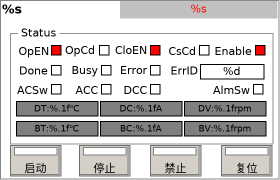
VISUALIZATION VPEModuleVis  // 280x180
VAR_IN_OUT
	userData: VPEHMIStruts;
END_VAR
    Button (10,145 51x31), "启动", input disabled if: NOT userData.HMIEnable
        tap userData.open
    Rectangle (14,147 43x8), colour toggle: userData.openRelay
    GroupBox (10,25 263x119), "Status"
        RoundedRectangle (41,40 10x10), colour toggle: userData.done
        RoundedRectangle (245,20 10x10), colour toggle: userData.enable
        RoundedRectangle (91,40 10x10), colour toggle: userData.busy
        RoundedRectangle (140,40 10x10), colour toggle: userData.error
        Rectangle (190,39 64x15), "%d", text variable: userData.errID
        Label (5,20 37x13), "OpEN"
        RoundedRectangle (41,20 10x10), colour toggle: userData.enableOpen
        RoundedRectangle (140,20 10x10), colour toggle: userData.enableClose
        Label (206,20 39x13), "Enable"
        Label (158,39 33x14), "ErrID"
        Label (110,39 30x13), "Error"
        Label (61,39 30x13), "Busy"
        Label (8,38 33x16), "Done"
        RoundedRectangle (41,59 10x10), colour toggle: userData.AccAprSw
        Label (203,59 40x13), "AlmSw"
        RoundedRectangle (243,59 10x10), colour toggle: userData.AlmAprSw
        Rectangle (6,96 82x15), "BT:%.1f℃", text variable: userData.BoosterTemperature, input disabled if: true
        RoundedRectangle (140,59 10x10), colour toggle: userData.Dccing
        RoundedRectangle (91,59 10x10), colour toggle: userData.Accing
        Label (52,19 36x13), "OpCd"
        RoundedRectangle (89,20 10x10), colour toggle: userData.opencondition
        Label (103,19 37x13), "CloEN"
    Button (221,145 51x31), "复位"
        tap userData.reset
    Rectangle (225,147 43x8), colour toggle: userData.reset
    Rectangle (-1,-1 119x20), "%s", text variable: userData.nameTXT
    Button (79,145 51x31), "停止"
        tap userData.close
    Rectangle (83,147 43x8)
    Label (14,84 37x13), "ACSw"
    Button (150,145 51x31), "禁止"
        tap userData.stop
    Rectangle (16,101 82x15), "DT:%.1f℃", text variable: userData.DryPumpTemperature, input disabled if: true
    Rectangle (100,101 82x15), "DC:%.1fA", text variable: userData.DryPumpCurrent, input disabled if: true
    Rectangle (184,101 82x15), "DV:%.1frpm", text variable: userData.DryPumpSpeed, input disabled if: true
    Rectangle (153,147 43x8)
    Rectangle (100,121 82x15), "BC:%.1fA", text variable: userData.BoosterCurrent, input disabled if: true
    Rectangle (184,121 82x15), "BV:%.1frpm", text variable: userData.BoosterSpeed, input disabled if: true
    Rectangle (120,0 157x18), "%s", text variable: userData.errTXT
    Label (113,84 37x13), "DCC"
    Label (70,84 31x13), "ACC"
    RoundedRectangle (199,45 10x10), colour toggle: userData.closecondition
    Label (165,45 34x13), "CsCd"
END_VISUALIZATION

(* stored: Version 1.1.0.1, ProductVersion 3.1.4024.4
   Visu VPEModuleVis: Id {eea821d3-db00-4871-8ac1-01b609a85683} *)
